FUNCTION_BLOCK GetDCTime
VAR_INPUT
END_VAR
VAR_OUTPUT
	actual	:	ULINT;
	tasktime	:	ULINT;
	ticktime	:	ULINT;
END_VAR
VAR
	aminustask	:	ULINT;
	aminustick	:	ULINT;
	taskminustick	:	ULINT;
	
	bb	:	BOOL;
	
	signalcomp :	SignalTimeComparison;
END_VAR

actual := F_GetActualDcTime64();
tasktime := F_GetCurDcTaskTime64();
ticktime := F_GetCurDcTickTime64();


// compares the offset to different dc time functions
IF bb THEN
	aminustask := actual - tasktime;
	aminustick := actual - ticktime;
	taskminustick := tasktime - ticktime;
	
	signalcomp(insignalTime := actual, outsignalTime := tasktime);
	
	bb := FALSE;
END_IF

END_FUNCTION_BLOCK

(* stored: Version 1.1.0.1, ProductVersion 3.1.4024.12
   POU GetDCTime: Id {8615e09d-95a9-42ce-988d-e0f5c8b259d9}, SpecialFunc None *)
